// TIA Portal V18 export
// export: Created 2026-06-08T16:32:21.0599713Z, ExportSetting WithDefaults, DisplayName Totally Integrated Automation Portal, DisplayVersion V18, DisplayName TIA Portal Openness, DisplayVersion V18, DisplayName TIA Portal Version Control Interface, DisplayVersion V18, DisplayName STEP 7 Professional, DisplayVersion V18, DisplayName STEP 7 Safety, DisplayVersion V18, DisplayName WinCC Professional, DisplayVersion V18
FUNCTION_BLOCK "BASE_execess_remove_station"   // FB7, LAD
VERSION : 0.1
// stored: AutoNumber true, IsIECCheckEnabled false, UDAEnableTagReadback false
BEGIN

REGION Network 1: LID_BELT_EXECESS_CONVYR_HANDLER
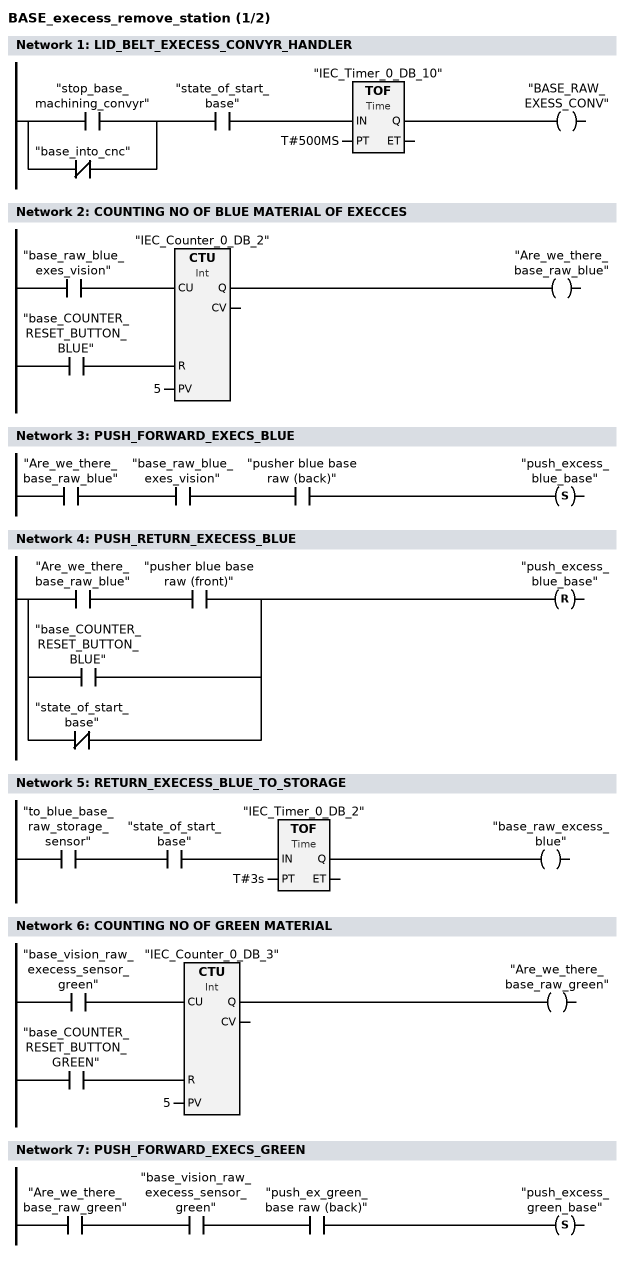
   RUNG wire#powerrail
      Contact( "stop_base_machining_convyr" )
      wire#w1
      Contact( "state_of_start_base" )
      { S7_Templates := "time_type := Time" } "IEC_Timer_0_DB_10".TOF(pt := T#500MS, et =>)
      Coil( "BASE_RAW_EXESS_CONV" )
   END_RUNG
   RUNG wire#powerrail
      I_Contact( "base_into_cnc" )
   END_RUNG wire#w1
   // the same network as SCL:
   "IEC_Timer_0_DB_10".TOF(IN := ("stop_base_machining_convyr" OR NOT "base_into_cnc") AND "state_of_start_base",
                           PT := T#500MS);
   "BASE_RAW_EXESS_CONV" := "IEC_Timer_0_DB_10".Q;
END_REGION

REGION Network 2: COUNTING NO OF BLUE MATERIAL OF EXECCES
   RUNG wire#powerrail
      Contact( "base_raw_blue_exes_vision" )
      { S7_Templates := "value_type := Int" } "IEC_Counter_0_DB_2".CTU(r := wire#w1, pv := 5, cv =>)
      Coil( "Are_we_there_base_raw_blue" )
   END_RUNG
   RUNG wire#powerrail
      Contact( "base_COUNTER_RESET_BUTTON_BLUE" )
   END_RUNG wire#w1
   // the same network as SCL:
   "IEC_Counter_0_DB_2".CTU(CU := "base_raw_blue_exes_vision", R := "base_COUNTER_RESET_BUTTON_BLUE", PV := 5);
   "Are_we_there_base_raw_blue" := "IEC_Counter_0_DB_2".Q;
END_REGION

REGION Network 3: PUSH_FORWARD_EXECS_BLUE
   RUNG wire#powerrail
      Contact( "Are_we_there_base_raw_blue" )
      Contact( "base_raw_blue_exes_vision" )
      Contact( "pusher blue base raw (back)" )
      S_Coil( "push_excess_blue_base" )
   END_RUNG
   // the same network as SCL:
   IF "Are_we_there_base_raw_blue" AND "base_raw_blue_exes_vision" AND "pusher blue base raw (back)" THEN
       "push_excess_blue_base" := TRUE;
   END_IF;
END_REGION

REGION Network 4: PUSH_RETURN_EXECESS_BLUE
   RUNG wire#powerrail
      Contact( "Are_we_there_base_raw_blue" )
      Contact( "pusher blue base raw (front)" )
      wire#w1
      R_Coil( "push_excess_blue_base" )
   END_RUNG
   RUNG wire#powerrail
      Contact( "base_COUNTER_RESET_BUTTON_BLUE" )
   END_RUNG wire#w1
   RUNG wire#powerrail
      I_Contact( "state_of_start_base" )
   END_RUNG wire#w1
   // the same network as SCL:
   IF ("Are_we_there_base_raw_blue" AND "pusher blue base raw (front)") OR "base_COUNTER_RESET_BUTTON_BLUE" OR NOT "state_of_start_base" THEN
       "push_excess_blue_base" := FALSE;
   END_IF;
END_REGION

REGION Network 5: RETURN_EXECESS_BLUE_TO_STORAGE
   RUNG wire#powerrail
      Contact( "to_blue_base_raw_storage_sensor" )
      Contact( "state_of_start_base" )
      { S7_Templates := "time_type := Time" } "IEC_Timer_0_DB_2".TOF(pt := T#3s, et =>)
      Coil( "base_raw_excess_blue" )
   END_RUNG
   // the same network as SCL:
   "IEC_Timer_0_DB_2".TOF(IN := "to_blue_base_raw_storage_sensor" AND "state_of_start_base", PT := T#3s);
   "base_raw_excess_blue" := "IEC_Timer_0_DB_2".Q;
END_REGION

REGION Network 6: COUNTING NO OF GREEN MATERIAL
   RUNG wire#powerrail
      Contact( "base_vision_raw_execess_sensor_green" )
      { S7_Templates := "value_type := Int" } "IEC_Counter_0_DB_3".CTU(r := wire#w1, pv := 5, cv =>)
      Coil( "Are_we_there_base_raw_green" )
   END_RUNG
   RUNG wire#powerrail
      Contact( "base_COUNTER_RESET_BUTTON_GREEN" )
   END_RUNG wire#w1
   // the same network as SCL:
   "IEC_Counter_0_DB_3".CTU(CU := "base_vision_raw_execess_sensor_green",
                           R := "base_COUNTER_RESET_BUTTON_GREEN",
                           PV := 5);
   "Are_we_there_base_raw_green" := "IEC_Counter_0_DB_3".Q;
END_REGION

REGION Network 7: PUSH_FORWARD_EXECS_GREEN
   RUNG wire#powerrail
      Contact( "Are_we_there_base_raw_green" )
      Contact( "base_vision_raw_execess_sensor_green" )
      Contact( "push_ex_green_base raw (back)" )
      S_Coil( "push_excess_green_base" )
   END_RUNG
   // the same network as SCL:
   IF "Are_we_there_base_raw_green" AND "base_vision_raw_execess_sensor_green" AND "push_ex_green_base raw (back)" THEN
       "push_excess_green_base" := TRUE;
   END_IF;
END_REGION

REGION Network 8: RETURN_EXECESS_GREEN_TO_STORAGE
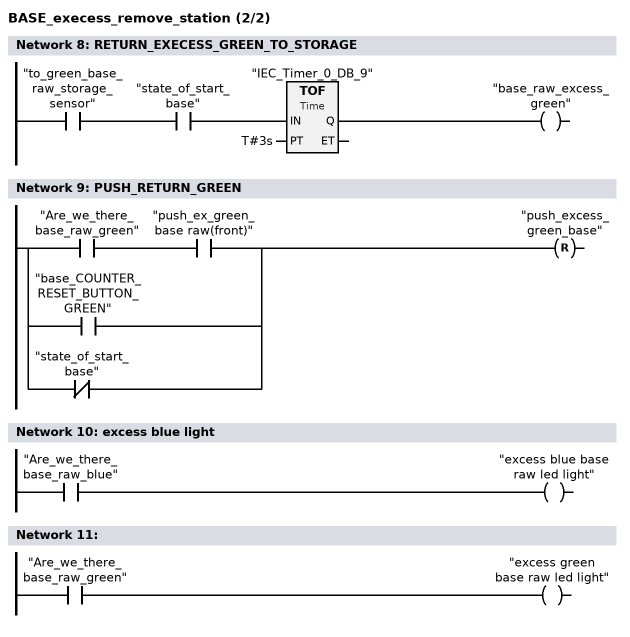
   RUNG wire#powerrail
      Contact( "to_green_base_raw_storage_sensor" )
      Contact( "state_of_start_base" )
      { S7_Templates := "time_type := Time" } "IEC_Timer_0_DB_9".TOF(pt := T#3s, et =>)
      Coil( "base_raw_excess_green" )
   END_RUNG
   // the same network as SCL:
   "IEC_Timer_0_DB_9".TOF(IN := "to_green_base_raw_storage_sensor" AND "state_of_start_base", PT := T#3s);
   "base_raw_excess_green" := "IEC_Timer_0_DB_9".Q;
END_REGION

REGION Network 9: PUSH_RETURN_GREEN
   RUNG wire#powerrail
      Contact( "Are_we_there_base_raw_green" )
      Contact( "push_ex_green_base raw(front)" )
      wire#w1
      R_Coil( "push_excess_green_base" )
   END_RUNG
   RUNG wire#powerrail
      Contact( "base_COUNTER_RESET_BUTTON_GREEN" )
   END_RUNG wire#w1
   RUNG wire#powerrail
      I_Contact( "state_of_start_base" )
   END_RUNG wire#w1
   // the same network as SCL:
   IF ("Are_we_there_base_raw_green" AND "push_ex_green_base raw(front)") OR "base_COUNTER_RESET_BUTTON_GREEN" OR NOT "state_of_start_base" THEN
       "push_excess_green_base" := FALSE;
   END_IF;
END_REGION

REGION Network 10: excess blue light
   RUNG wire#powerrail
      Contact( "Are_we_there_base_raw_blue" )
      Coil( "excess blue base raw led light" )
   END_RUNG
   // the same network as SCL:
   "excess blue base raw led light" := "Are_we_there_base_raw_blue";
END_REGION

REGION Network 11
   RUNG wire#powerrail
      Contact( "Are_we_there_base_raw_green" )
      Coil( "excess green base raw led light" )
   END_RUNG
   // the same network as SCL:
   "excess green base raw led light" := "Are_we_there_base_raw_green";
END_REGION
END_FUNCTION_BLOCK
